FUNCTION_BLOCK SPLIT_AL_INTO_AW (* this Function splits the 4 AW (WORD) adapters from a AL (LWORD) *)
  (* Standard: 61499-2; Description: Copyright (c) 2026 Meisterschulen am Ostbahnhof SPDX-License-Identifier: EPL-2.0 *)
  (* Version 1.0, 2026-05-16, Franz Höpfinger, Meisterschulen am Ostbahnhof, initial API and implementation and/or initial documentation *)
  PACKAGE adapter::splitting;
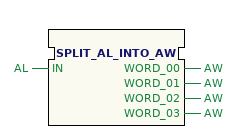
  SOCKETS
    IN : adapter::types::unidirectional::AL; (* LWORD Input *)
  END_SOCKETS
  PLUGS
    WORD_00 : adapter::types::unidirectional::AW; (* Word 0 *)
    WORD_01 : adapter::types::unidirectional::AW; (* Word 1 *)
    WORD_02 : adapter::types::unidirectional::AW; (* Word 2 *)
    WORD_03 : adapter::types::unidirectional::AW; (* Word 3 *)
  END_PLUGS
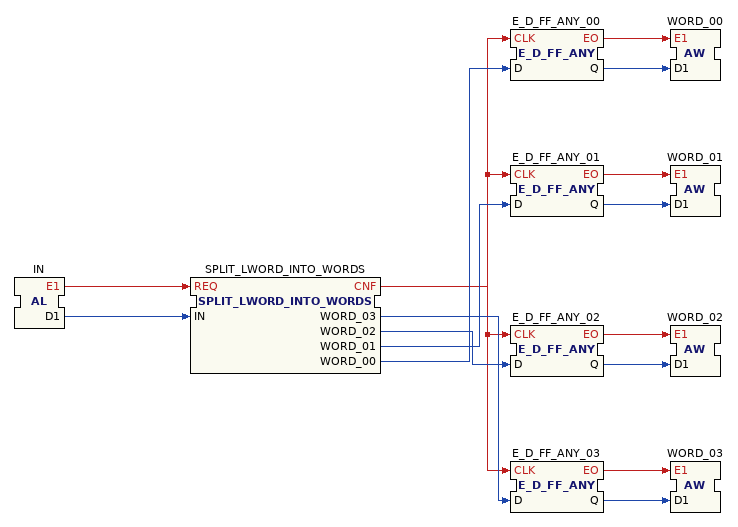
  FBS
    E_D_FF_ANY_00 : iec61499::events::E_D_FF_ANY;
    E_D_FF_ANY_01 : iec61499::events::E_D_FF_ANY;
    E_D_FF_ANY_02 : iec61499::events::E_D_FF_ANY;
    E_D_FF_ANY_03 : iec61499::events::E_D_FF_ANY;
    SPLIT_LWORD_INTO_WORDS : eclipse4diac::utils::splitting::SPLIT_LWORD_INTO_WORDS;
  END_FBS
  EVENT_CONNECTIONS
    IN.E1 TO SPLIT_LWORD_INTO_WORDS.REQ;
    SPLIT_LWORD_INTO_WORDS.CNF TO E_D_FF_ANY_00.CLK;
    SPLIT_LWORD_INTO_WORDS.CNF TO E_D_FF_ANY_01.CLK;
    SPLIT_LWORD_INTO_WORDS.CNF TO E_D_FF_ANY_02.CLK;
    SPLIT_LWORD_INTO_WORDS.CNF TO E_D_FF_ANY_03.CLK;
    E_D_FF_ANY_00.EO TO WORD_00.E1;
    E_D_FF_ANY_01.EO TO WORD_01.E1;
    E_D_FF_ANY_02.EO TO WORD_02.E1;
    E_D_FF_ANY_03.EO TO WORD_03.E1;
  END_CONNECTIONS
  DATA_CONNECTIONS
    IN.D1 TO SPLIT_LWORD_INTO_WORDS.IN;
    SPLIT_LWORD_INTO_WORDS.WORD_03 TO E_D_FF_ANY_03.D;
    SPLIT_LWORD_INTO_WORDS.WORD_02 TO E_D_FF_ANY_02.D;
    SPLIT_LWORD_INTO_WORDS.WORD_01 TO E_D_FF_ANY_01.D;
    SPLIT_LWORD_INTO_WORDS.WORD_00 TO E_D_FF_ANY_00.D;
    E_D_FF_ANY_00.Q TO WORD_00.D1;
    E_D_FF_ANY_01.Q TO WORD_01.D1;
    E_D_FF_ANY_02.Q TO WORD_02.D1;
    E_D_FF_ANY_03.Q TO WORD_03.D1;
  END_CONNECTIONS
END_FUNCTION_BLOCK
